// TIA Portal project "Project5" (V17)

(* hardware
DEVICE "S7-1200 station_1"  S7-1200 Station
   slot 0: "Rack_0"  S7-1200 Rack  Rack  V1.0
   slot 1: "PLC_1"  CPU 1214C AC/DC/Rly  6ES7 214-1BG40-0XB0  V4.2
*)

// ===== PLC "PLC_1"  CPU 1214C AC/DC/Rly =====

VAR_GLOBAL   // PLC tag table "Default tag table"
   "PB1" AT %I0.0 : Bool;
   "PB2" AT %I0.1 : Bool;
   "X1" AT %M0.0 : Bool;
   "X2" AT %M0.1 : Bool;
   "PL1" AT %Q0.0 : Bool;
   "PL2" AT %Q0.1 : Bool;
   "Tag_1" AT %MD100 : Time;
END_VAR

// folder: System blocks/Program resources

DATA_BLOCK "T1"   // DB1
{ S7_Optimized_Access := 'TRUE' }
AUTHOR : Simatic
FAMILY : IEC
NAME : IEC_TMR
VERSION : 1.0
// stored: InstanceOfName IEC_TIMER
"IEC_TIMER"
BEGIN
END_DATA_BLOCK

DATA_BLOCK "T2"   // DB2
{ S7_Optimized_Access := 'TRUE' }
AUTHOR : Simatic
FAMILY : IEC
NAME : IEC_TMR
VERSION : 1.0
// stored: InstanceOfName IEC_TIMER
"IEC_TIMER"
BEGIN
END_DATA_BLOCK

// folder: (top level)

ORGANIZATION_BLOCK "Main"   // OB1, LAD, ProgramCycle
TITLE = "Main Program Sweep (Cycle)"
{ S7_Optimized_Access := 'TRUE' }
VERSION : 0.1
   VAR_INPUT
      Initial_Call : Bool;   // Initial call of this OB
      Remanence : Bool;   // =True, if remanent data are available
   END_VAR
BEGIN

REGION Network 1
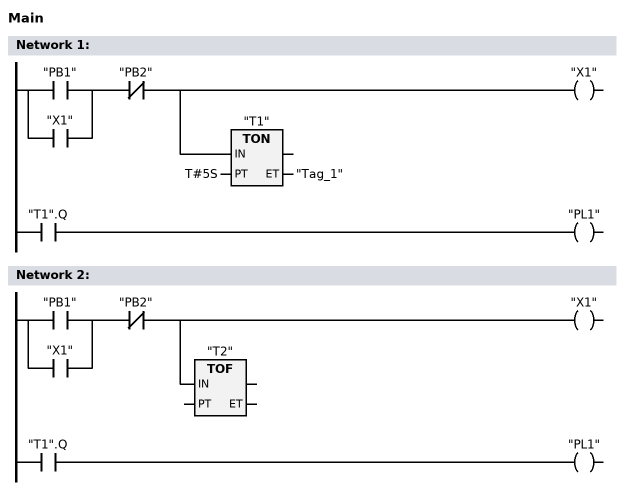
   "X1" := ("PB1" OR "X1") AND NOT "PB2";
   "T1".TON(IN := "X1", PT := T#5S, ET => "Tag_1");
   "PL1" := "T1".Q;
END_REGION

REGION Network 2
   "X1" := ("PB1" OR "X1") AND NOT "PB2";
   "T2".TOF(IN := "X1");
   "PL1" := "T1".Q;
END_REGION
END_ORGANIZATION_BLOCK